FUNCTION_BLOCK AUDI_SPLIT_2 (* SPLIT 1 AUDI into 2 AUDI (generic FB) Adapter-Ausgang wird nur bei Wertänderung aktualisiert (Event nur bei tatsächlicher Änderung). *)
  (* Standard: 61499-2; Description: Copyright (c) 2025 HR Agrartechnik GmbH This program and the accompanying materials are made available under the terms of the Eclipse Public License 2.0 which is available at https://www.eclipse.org/legal/epl-2.0/ SPDX-License-Identifier: EPL-2.0 *)
  (* Version 1.0, 2025-01-24, Franz Höpfinger, HR Agrartechnik GmbH *)
  PACKAGE adapter::events::unidirectional;
  IMPORT eclipse4diac::core::GenericClassName;
  {SET_ATTRIBUTE(eclipse4diac::core::GenericClassName, 'GEN_AUDI_SPLIT')}
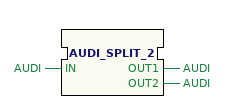
  SOCKETS
    IN : adapter::types::unidirectional::AUDI;
  END_SOCKETS
  PLUGS
    OUT1 : adapter::types::unidirectional::AUDI;
    OUT2 : adapter::types::unidirectional::AUDI;
  END_PLUGS
END_FUNCTION_BLOCK
